// TwinCAT 3 PLC project PLC
// ProgramVersion: 3.1.4024.0
// libraries:
//   Tc2_Standard, * (Beckhoff Automation GmbH)
//   Tc2_System, * (Beckhoff Automation GmbH)
//   Tc3_Module, * (Beckhoff Automation GmbH)
// project tree:
//   / PlcTask.TcTTO
//   POUs/ MAIN.TcPOU, PumpControl.TcPOU
// real-time tasks:
//   TASK PlcTask: cycle T#10ms, priority 20, ADS port 350

CONFIGURATION PLC
    RESOURCE PLC ON TwinCAT3
        TASK PlcTask(INTERVAL := T#10ms, PRIORITY := 20);
        PROGRAM MAIN WITH PlcTask : MAIN;
    END_RESOURCE
END_CONFIGURATION

// ---- POUs/MAIN.TcPOU
PROGRAM MAIN
VAR_INPUT
END_VAR
VAR_OUTPUT
END_VAR
VAR
	Pump01						: PumpControl;
	ManAutoPb					: BOOL;
	ManPumpStart				: BOOL;						// N.O.
	ManPumpStop					: BOOL := TRUE;				// N.C.
	LevelSensorMin				: BOOL := TRUE;				// N.C.
	LevelSensorMax				: BOOL := TRUE;				// N.C.
	PumpRunning					: BOOL;
	ManAutoState				: BOOL;
END_VAR

Pump01(
    ManAutoPb := ManAutoPb,
    ManPumpStart := ManPumpStart,
    ManPumpStop := ManPumpStop,
    LevelSensorMin := LevelSensorMin,
    LevelSensorMax := LevelSensorMax); // PumpControl
PumpRunning := Pump01.PumpRunning;
ManAutoState := Pump01.ManAutoState;

END_PROGRAM

// ---- POUs/PumpControl.TcPOU
FUNCTION_BLOCK PumpControl
VAR_INPUT
	ManAutoPb			:	BOOL;			// Manual / auto mode; TRUE=Manual
	ManPumpStart		:	BOOL;			// Command Pump On in Manual Mode (N.O.)
	ManPumpStop			:	BOOL;			// Command Pump Off in Manual Mode (N.C)
	LevelSensorMin		:	BOOL;			// Tank low level sensor (N.C)
	LevelSensorMax		:	BOOL;			// Tank high level sensor (N.C)
END_VAR
VAR_OUTPUT
	PumpRunning			:	BOOL;			// Motor pump RUN state
	ManAutoState		:	BOOL;			// Indication of manual / auto mode
END_VAR
VAR
	srPumpRunning		: SR;
	PumpOffCommand		: BOOL;
	tonDelay			: TON;
	rtrigManAuto		: R_TRIG;
END_VAR

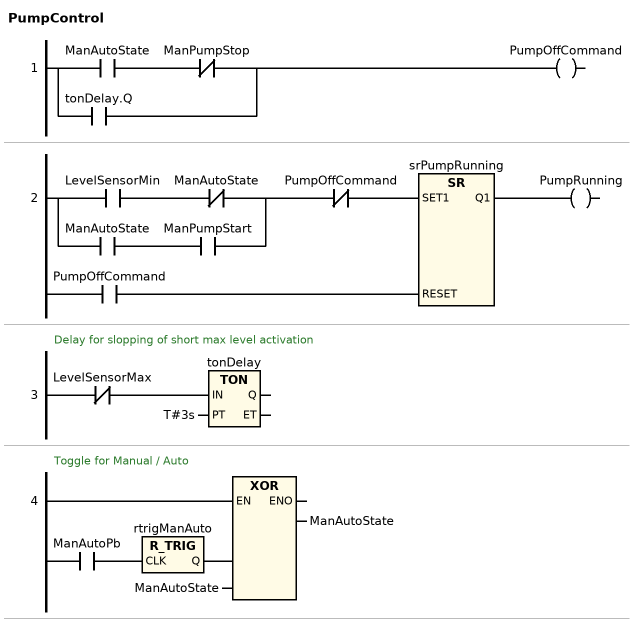
// NETWORK 1
PumpOffCommand := ManAutoState AND NOT ManPumpStop OR tonDelay.Q;

// NETWORK 2
srPumpRunning(SET1 := (LevelSensorMin AND NOT ManAutoState OR ManAutoState AND ManPumpStart) AND NOT PumpOffCommand, RESET := PumpOffCommand); // SR
PumpRunning := srPumpRunning.Q1;

// NETWORK 3
// Delay for slopping of short max level activation
tonDelay(IN := NOT LevelSensorMax, PT := T#3s); // TON

// NETWORK 4
// Toggle for Manual / Auto
rtrigManAuto(CLK := ManAutoPb); // R_TRIG
ManAutoState := rtrigManAuto.Q XOR ManAutoState;

END_FUNCTION_BLOCK
